PROGRAM Home
VAR
	SimsX_Home: MC_MoveAbsolute;
	SimsX_Home_ErrorID: UDINT;
	SimsY_Home: MC_MoveAbsolute;
	SimsZ_Home: MC_MoveAbsolute;
	SimsY_Home_ErrorID: UDINT;
	SimsZ_Home_ErrorID: UDINT;
	Inside_Dia: LREAL;
	Pos_Exists: BOOL;
	Pos_NotValid: BOOL;
END_VAR

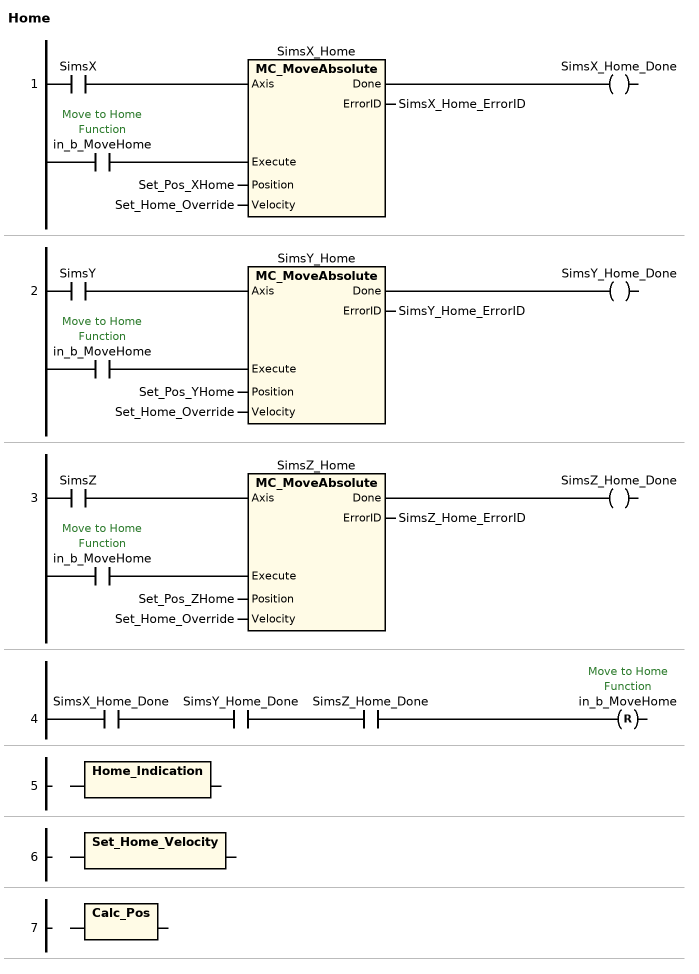
// NETWORK 1
//   in_b_MoveHome: Move to Home Function
SimsX_Home(
    Axis := SimsX,
    Execute := in_b_MoveHome,
    Position := Set_Pos_XHome,
    Velocity := Set_Home_Override,
    ErrorID => SimsX_Home_ErrorID); // MC_MoveAbsolute
SimsX_Home_Done := SimsX_Home.Done;

// NETWORK 2
//   in_b_MoveHome: Move to Home Function
SimsY_Home(
    Axis := SimsY,
    Execute := in_b_MoveHome,
    Position := Set_Pos_YHome,
    Velocity := Set_Home_Override,
    ErrorID => SimsY_Home_ErrorID); // MC_MoveAbsolute
SimsY_Home_Done := SimsY_Home.Done;

// NETWORK 3
//   in_b_MoveHome: Move to Home Function
SimsZ_Home(
    Axis := SimsZ,
    Execute := in_b_MoveHome,
    Position := Set_Pos_ZHome,
    Velocity := Set_Home_Override,
    ErrorID => SimsZ_Home_ErrorID); // MC_MoveAbsolute
SimsZ_Home_Done := SimsZ_Home.Done;

// NETWORK 4
//   in_b_MoveHome: Move to Home Function
in_b_MoveHome R= SimsX_Home_Done AND SimsY_Home_Done AND SimsZ_Home_Done;

// NETWORK 5
Home_Indication();

// NETWORK 6
Set_Home_Velocity();

// NETWORK 7
Calc_Pos();

ACTION Calc_Pos:
Inside_Dia:= SQRT((Set_Pos_XHome)*(Set_Pos_XHome)+
				  (Set_Pos_YHome)*(Set_Pos_YHome));
				  
IF Inside_Dia>=251 OR Set_Pos_ZHome>=70 OR Set_Pos_ZHome<=-160 THEN
	Pos_Exists:=FALSE;	
	Pos_NotValid:=TRUE;
ELSE
	Pos_Exists:=TRUE;
	Pos_NotValid:=FALSE;
END_IF
END_ACTION

ACTION Home_Indication:
IF (Set_Pos_XHome <= (SimsX.NcToPlc.ActPos+0.5) AND  Set_Pos_XHome >= (SimsX.NcToPlc.ActPos-0.5)) AND
   (Set_Pos_YHome <= (SimsY.NcToPlc.ActPos+0.5) AND  Set_Pos_YHome >= (SimsY.NcToPlc.ActPos-0.5)) AND
   (Set_Pos_ZHome <= (SimsZ.NcToPlc.ActPos+0.5) AND  Set_Pos_ZHome >= (SimsZ.NcToPlc.ActPos-0.5))
 THEN
	out_b_inHome := TRUE;
ELSE
	out_b_inHome := FALSE;
END_IF
END_ACTION

ACTION Set_Home_Velocity:

Set_Home_Override := (Set_Home_Override*(in_uiMasterAxes_Override/100));
END_ACTION

END_PROGRAM

(* stored: Version 1.1.0.1, ProductVersion 3.1.4018.9
   POU Home: Id {a045509a-ee3a-4de5-a82b-add5e08a861e}, SpecialFunc None
   Action Calc_Pos: Id {1548b73e-b2b4-432e-af2c-9ac6f3057bff}
   Action Home_Indication: Id {96b09bb5-1c4e-43a8-b9be-8f4ff4409875}
   Action Set_Home_Velocity: Id {c5a8541e-2142-4b5b-8ed5-22f473abefa2} *)
